{attribute addProperty BoxType "AT2050-0501-0017"}
{attribute addProperty Id "A_0088_AT2050_5501_0017_AT2050_5501AT2050_C5E5984862678.25"}
{attribute addProperty CRC "1595119970"}
{attribute addProperty SizeInBites "626"}
{attribute addProperty SizeInBytes "78.25"}
TYPE A_0056_AT2050_0501_0017_5F139962 EXTENDS AT2050_BA5A9548 :
STRUCT
	{attribute addProperty Name "A_0088_AT2050_5501_0017_AT2050_5501"}
	A_0088_AT2050_5501_0017_AT2050_5501 : AT2050_C5E59848;
END_STRUCT
END_TYPE

(* stored: Version 1.2.0.0, ProductVersion 3.1.4024.9
   DUT A_0056_AT2050_0501_0017_5F139962: Id {30945328-a102-407c-8487-7028eda2332a} *)
